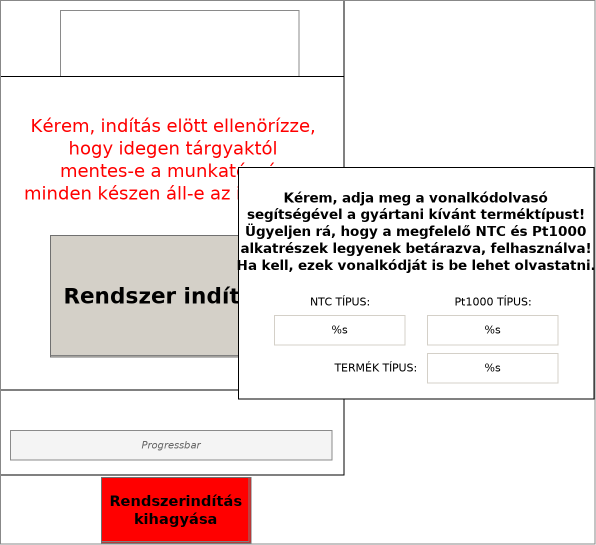
VISUALIZATION Start_ablak  // 596x545
    RoundedRectangle (0,0 344x475)
    Group (0,10 594x533)
        Frame (60,0 239x320)
            shows Start_ellenorzes()
        Group (0,66 344x314), invisible if: INIT.iState>0
            RoundedRectangle (0,0 344x314), invisible if: INIT.iState>0, input disabled if: INIT.iState>0
            Label (13,21 320x125), "Kérem, indítás elött ellenörízze, hogy idegen tárgyaktól mentes-e a munkatér, és minden készen áll-e az indításra!"
            Button (50,159 246x122), "Rendszer indítása", invisible if: INIT.iState>0, input disabled if: INIT.iState>0
                OnMouseClick: execute { INIT.iState:=1; }
        Button (101,467 150x66), "Rendszerindítás kihagyása"
            OnMouseClick: execute {
                INIT.iState:=5;
                GVL.bSystemStarted:=TRUE;
                GVL.bSystemNotStarted:=FALSE;
            }
        Progressbar (10,420 322x30), variable: INIT.iKeszenletFoka, invisible if: GVL.bSystemStarted
        Group (238,157 356x232), invisible if: NOT INIT.bLezerKesz
            RoundedRectangle (0,0 356x232)
            Group (36,125 284x91), invisible if: NOT INIT.bLezerKesz
                Label (11,0 110x20), "NTC TÍPUS:"
                Textfield (0,23 131x30), "%s", text variable: GVL.sNTCTypeElozo, colour toggle: GVL.sNTCType='HIBÁS KÓD'
                    OnMouseClick: write GVL.sNTCType via Edit
                Textfield (153,23 131x30), "%s", text variable: GVL.sPtTypeElozo, colour toggle: GVL.sPtType='HIBÁS KÓD'
                    OnMouseClick: write GVL.sPtType via Edit
                Label (164,0 110x20), "Pt1000 TÍPUS:"
                Group (47,61 237x30)
                    Textfield (106,0 131x30), "%s", text variable: GVL.sProductType, colour toggle: NOT GVL.bProductTypeOK
                        OnMouseClick: write the text variable via Edit
                    Label (0,5 110x20), "TERMÉK TÍPUS:"
            Label (8,13 340x103), "Kérem, adja meg a vonalkódolvasó segítségével a gyártani kívánt terméktípust! Ügyeljen rá, hogy a megfelelő NTC és Pt1000 alkatrészek legyenek betárazva, felhasználva! Ha kell, ezek vonalkódját is be lehet olvastatni."
END_VISUALIZATION

(* stored: Version 1.1.0.1, ProductVersion 3.1.4024.11
   Visu Start_ablak: Id {1b9e66d6-0a8e-418e-90dd-a4f606e3d314} *)
